(* IEC 61131-3 sources: wts-100-water-treatment-skid/plc, 4 files *)

(* ---- POU_ALARMS.st ---- *)
(*
    WTS-100  POU_ALARMS
    Alarm management.  IEC 61131-3 Structured Text.

    Implements section 6 of the control narrative, to ISA-18.2.

    FIRST OUT
    One fault usually sets off several alarms.  Supply fails, so the pump
    stops, so flow falls, so level drops, so temperature deviates.  Five
    alarms, one cause.  FIRST_OUT records whichever came first while no alarm
    was already standing, because that is the one that actually broke.
    Without it an operator at 3 a.m. faces a screen of alarms with no way to
    tell cause from consequence.

    PRIORITY
    Set by consequence and by how fast the operator must react.
    If everything is critical then nothing is.
*)

FUNCTION_BLOCK POU_ALARMS

VAR_INPUT
    ESD_01_OK       : BOOL;
    TSHH_102_OK     : BOOL;
    LSHH_102_OK     : BOOL;
    LSLL_101_OK     : BOOL;
    BOTH_PUMPS_FAIL : BOOL;
    DUTY_CHANGEOVER : BOOL;
    AIN_INVALID     : BOOL;
    AIN_STUCK       : BOOL;
    SEQ_TIMEOUT     : BOOL;
    TEMP_DEVIATION  : BOOL;
    PUMP_FB_MISMATCH: BOOL;
    DOSE_DEVIATION  : BOOL;
    ACK_CMD         : BOOL;
END_VAR

VAR_OUTPUT
    ALM_001 : BOOL;   (* emergency stop            Critical *)
    ALM_002 : BOOL;   (* over temperature          Critical *)
    ALM_003 : BOOL;   (* both raw pumps failed     Critical *)
    ALM_004 : BOOL;   (* treatment tank too full   High     *)
    ALM_005 : BOOL;   (* raw tank empty            High     *)
    ALM_006 : BOOL;   (* duty pump failed          High     *)
    ALM_007 : BOOL;   (* analog signal bad         High     *)
    ALM_008 : BOOL;   (* signal not changing       Medium   *)
    ALM_009 : BOOL;   (* sequence timeout          Medium   *)
    ALM_010 : BOOL;   (* temperature deviation     Medium   *)
    ALM_011 : BOOL;   (* pump feedback mismatch    Medium   *)
    ALM_012 : BOOL;   (* dosing deviation          Low      *)

    ANY_ALARM       : BOOL;
    ANY_UNACK       : BOOL;
    FIRST_OUT_ID    : INT;    (* 0 none, else 1..12 *)
    HIGHEST_PRIORITY: INT;    (* 0 none, 1 Critical, 2 High, 3 Medium, 4 Low *)
    ALM_HORN        : BOOL;
    ALM_BEACON      : BOOL;
END_VAR

VAR
    acked       : BOOL;
    prev_any    : BOOL;
    beacon_tick : TON;
END_VAR

(* --- alarm conditions --------------------------------------------------- *)
ALM_001 := NOT ESD_01_OK;
ALM_002 := NOT TSHH_102_OK;
ALM_003 := BOTH_PUMPS_FAIL;
ALM_004 := NOT LSHH_102_OK;
ALM_005 := NOT LSLL_101_OK;
ALM_006 := DUTY_CHANGEOVER;
ALM_007 := AIN_INVALID;
ALM_008 := AIN_STUCK;
ALM_009 := SEQ_TIMEOUT;
ALM_010 := TEMP_DEVIATION;
ALM_011 := PUMP_FB_MISMATCH;
ALM_012 := DOSE_DEVIATION;

ANY_ALARM := ALM_001 OR ALM_002 OR ALM_003 OR ALM_004 OR ALM_005 OR ALM_006
          OR ALM_007 OR ALM_008 OR ALM_009 OR ALM_010 OR ALM_011 OR ALM_012;

(* --- first out.
   --- Only captured when nothing was already standing, otherwise a later
   --- consequence would overwrite the real root cause.                  --- *)
IF ANY_ALARM AND (FIRST_OUT_ID = 0) THEN
    IF      ALM_001 THEN FIRST_OUT_ID := 1;
    ELSIF   ALM_002 THEN FIRST_OUT_ID := 2;
    ELSIF   ALM_003 THEN FIRST_OUT_ID := 3;
    ELSIF   ALM_004 THEN FIRST_OUT_ID := 4;
    ELSIF   ALM_005 THEN FIRST_OUT_ID := 5;
    ELSIF   ALM_006 THEN FIRST_OUT_ID := 6;
    ELSIF   ALM_007 THEN FIRST_OUT_ID := 7;
    ELSIF   ALM_008 THEN FIRST_OUT_ID := 8;
    ELSIF   ALM_009 THEN FIRST_OUT_ID := 9;
    ELSIF   ALM_010 THEN FIRST_OUT_ID := 10;
    ELSIF   ALM_011 THEN FIRST_OUT_ID := 11;
    ELSIF   ALM_012 THEN FIRST_OUT_ID := 12;
    END_IF;
END_IF;

IF NOT ANY_ALARM THEN
    FIRST_OUT_ID := 0;
END_IF;

(* --- highest standing priority ------------------------------------------ *)
IF   ALM_001 OR ALM_002 OR ALM_003                        THEN HIGHEST_PRIORITY := 1;
ELSIF ALM_004 OR ALM_005 OR ALM_006 OR ALM_007            THEN HIGHEST_PRIORITY := 2;
ELSIF ALM_008 OR ALM_009 OR ALM_010 OR ALM_011            THEN HIGHEST_PRIORITY := 3;
ELSIF ALM_012                                             THEN HIGHEST_PRIORITY := 4;
ELSE                                                           HIGHEST_PRIORITY := 0;
END_IF;

(* --- acknowledge.
   --- A NEW alarm clears the acknowledgement, so the horn sounds again
   --- rather than staying silent because an earlier one was acked.      --- *)
IF ANY_ALARM AND NOT prev_any THEN
    acked := FALSE;
END_IF;
prev_any := ANY_ALARM;

IF ACK_CMD THEN
    acked := TRUE;
END_IF;

IF NOT ANY_ALARM THEN
    acked := FALSE;
END_IF;

ANY_UNACK := ANY_ALARM AND NOT acked;

(* --- annunciation.
   --- Horn on any unacknowledged alarm.
   --- Beacon flashes while unacknowledged, steady once acked but still
   --- standing, so a glance tells you both things at once.              --- *)
ALM_HORN := ANY_UNACK;

beacon_tick(IN := NOT beacon_tick.Q, PT := T#500ms);
IF ANY_UNACK THEN
    ALM_BEACON := beacon_tick.Q;
ELSIF ANY_ALARM THEN
    ALM_BEACON := TRUE;
ELSE
    ALM_BEACON := FALSE;
END_IF;

END_FUNCTION_BLOCK

(* ---- POU_PUMPS.st ---- *)
(*
    WTS-100  POU_PUMPS
    Duty and standby raw water pumps.  IEC 61131-3 Structured Text.

    Same logic as the ladder drawing drawings/ladder_pumps.svg.

    Logic verified by test_ladder.py, 10 cases.
*)

FUNCTION_BLOCK POU_PUMPS

VAR_INPUT
    HS_02_START     : BOOL;   (* start pushbutton, momentary NO   *)
    HS_03_STOP_OK   : BOOL;   (* stop pushbutton, wired NC        *)
    PERM_RAW_PUMPS  : BOOL;   (* from POU_SAFETY                  *)
    XS_101A         : BOOL;   (* pump A run feedback              *)
    XS_101B         : BOOL;   (* pump B run feedback              *)
    BATCH_DONE      : BOOL;   (* one shot at end of a batch       *)
END_VAR

VAR_OUTPUT
    MTR_101A            : BOOL;
    MTR_101B            : BOOL;
    RUN_REQ             : BOOL;
    FAULT_A             : BOOL;
    FAULT_B             : BOOL;
    BOTH_PUMPS_FAILED   : BOOL;
    DUTY_IS_A           : BOOL := TRUE;
END_VAR

VAR
    tA          : TON;
    tB          : TON;
    batch_prev  : BOOL;
END_VAR

(* --- RUNG 1  start and stop with seal in.
   --- The seal in parallels the START contact ONLY.  Stop and the safety
   --- permission stay in series after it, so both can always break the rung.
   --- Putting them inside the seal in would mean the stop button does not
   --- stop the pumps once they are running.                              --- *)
RUN_REQ := (HS_02_START OR RUN_REQ) AND HS_03_STOP_OK AND PERM_RAW_PUMPS;

(* --- duty alternation.  Swap on each completed batch so running hours
   --- stay even between the two pumps.                                   --- *)
IF BATCH_DONE AND NOT batch_prev THEN
    DUTY_IS_A := NOT DUTY_IS_A;
END_IF;
batch_prev := BATCH_DONE;

(* --- RUNG 2  duty pump A                                               --- *)
MTR_101A := RUN_REQ AND DUTY_IS_A AND NOT FAULT_A;

(* --- RUNG 3  standby pump B.  Runs when B is duty, or when A has failed --- *)
MTR_101B := RUN_REQ AND NOT FAULT_B AND ((NOT DUTY_IS_A) OR FAULT_A);

(* --- RUNG 4 and 5  fault detection.
   --- Commanded on but no run feedback within 3 s means the motor did not
   --- actually start: tripped overload, failed contactor, blown fuse.    --- *)
tA(IN := MTR_101A AND NOT XS_101A, PT := T#3s);
tB(IN := MTR_101B AND NOT XS_101B, PT := T#3s);

IF tA.Q THEN FAULT_A := TRUE; END_IF;
IF tB.Q THEN FAULT_B := TRUE; END_IF;

(* --- RUNG 6  both pumps failed.  Interlock I6, trips the plant.        --- *)
BOTH_PUMPS_FAILED := FAULT_A AND FAULT_B;

END_FUNCTION_BLOCK

(* ---- POU_SAFETY.st ---- *)
(*
    WTS-100  POU_SAFETY
    Interlocks and permissives.  IEC 61131-3 Structured Text.

    This is the same logic as the ladder drawing drawings/ladder_safety.svg, written as
    text so it can be pasted straight into OpenPLC Editor and compiled.

    Runs FIRST in the scan, before the sequence and the loops, so nothing
    downstream can command an output this block has inhibited.

    All discrete safety contacts are wired normally closed.  Healthy = TRUE.
    A broken wire reads FALSE and therefore trips.

    Logic verified by test_ladder.py, 16 cases.
*)

FUNCTION_BLOCK POU_SAFETY

VAR_INPUT
    ESD_01_OK       : BOOL;   (* emergency stop not pressed      *)
    TSHH_102_OK     : BOOL;   (* below the 85 degC thermostat    *)
    XA_101A_OK      : BOOL;   (* pump A overload healthy         *)
    XA_101B_OK      : BOOL;   (* pump B overload healthy         *)
    LSLL_101_OK     : BOOL;   (* raw tank not at low low         *)
    LSHH_102_OK     : BOOL;   (* treat tank not at high high     *)
    LT_102_VALID    : BOOL;   (* level reading trustworthy       *)
    TT_102_VALID    : BOOL;   (* temperature reading trustworthy *)
    LT_102_MM       : REAL;   (* scaled treatment tank level     *)
    HS_04_RESET     : BOOL;   (* reset pushbutton                *)
END_VAR

VAR_OUTPUT
    PERM_RAW_PUMPS  : BOOL;
    PERM_HEATER     : BOOL;
    PERM_INLET      : BOOL;
    TRIP            : BOOL;
    TRIP_CAUSE      : BOOL;
    FIRST_OUT       : INT;    (* 0 none, else the interlock number *)
END_VAR

VAR
    ain_timer   : TON;
    AIN_FAULT   : BOOL;
    LVL_OK      : BOOL;
END_VAR

VAR CONSTANT
    LVL_HEATER_MIN : REAL := 800.0;
END_VAR

(* --- analog fault, interlock I7.  30 s so a brief glitch is ridden out --- *)
ain_timer(IN := NOT (LT_102_VALID AND TT_102_VALID), PT := T#30s);
AIN_FAULT := ain_timer.Q;

LVL_OK := (LT_102_MM >= LVL_HEATER_MIN);

(* --- RUNG 1  trip causes.  These are ALTERNATIVES, so OR not AND.       ---
   --- The two pump overloads are ANDed, because one failed pump changes  ---
   --- over to the standby and does not trip the plant.                   --- *)
TRIP_CAUSE :=  (NOT ESD_01_OK)
            OR (NOT TSHH_102_OK)
            OR ((NOT XA_101A_OK) AND (NOT XA_101B_OK))
            OR AIN_FAULT;

(* --- RUNG 2 and 3  latch and reset.
   --- Reset only clears the trip when the cause has already gone.        --- *)
IF TRIP_CAUSE THEN
    TRIP := TRUE;
    IF FIRST_OUT = 0 THEN
        IF    NOT ESD_01_OK                             THEN FIRST_OUT := 1;
        ELSIF NOT TSHH_102_OK                           THEN FIRST_OUT := 4;
        ELSIF (NOT XA_101A_OK) AND (NOT XA_101B_OK)     THEN FIRST_OUT := 6;
        ELSIF AIN_FAULT                                 THEN FIRST_OUT := 7;
        END_IF;
    END_IF;
ELSIF HS_04_RESET THEN
    TRIP      := FALSE;
    FIRST_OUT := 0;
END_IF;

(* --- RUNG 4  permission to run the raw water pumps.  I2 and I3.        --- *)
PERM_RAW_PUMPS := ESD_01_OK AND LSLL_101_OK AND LSHH_102_OK AND NOT TRIP;

(* --- RUNG 5  permission to run the heater.  I4 and I5.
   --- The level test uses the MEASURED level, never the sequence state,  ---
   --- so a defect in the sequence cannot fire a dry element.             --- *)
PERM_HEATER := ESD_01_OK AND TSHH_102_OK AND LT_102_VALID
               AND TT_102_VALID AND LVL_OK AND NOT TRIP;

(* --- RUNG 6  permission to open the inlet.  I3.                        --- *)
PERM_INLET := ESD_01_OK AND LSHH_102_OK AND NOT TRIP;

END_FUNCTION_BLOCK

(* ---- POU_SEQUENCE.st ---- *)
(*
    WTS-100  POU_SEQUENCE
    Batch sequence.  IEC 61131-3 Structured Text.

    IDLE -> FILL -> HEAT -> HOLD -> DISCHARGE -> DRAIN -> IDLE

    One state is active at a time.  Every transition out of every state is
    listed.  Every state has a timeout, because a state machine with no
    timeout can wait forever for a condition that will never arrive, and the
    operator gets no indication why nothing is happening.

    Any interlock forces TRIP from any state.  TRIP is latched.

    Implements section 4 of the control narrative.
*)

FUNCTION_BLOCK POU_SEQUENCE

VAR_INPUT
    START_CMD       : BOOL;
    HOLD_CMD        : BOOL;
    ABORT_CMD       : BOOL;
    AUTO_MODE       : BOOL;
    TRIP            : BOOL;     (* from POU_SAFETY *)
    PERM_INLET      : BOOL;
    PERM_HEATER     : BOOL;
    LT_101_MM       : REAL;
    LT_102_MM       : REAL;
    TT_102_C        : REAL;
    TEMP_SETPOINT   : REAL;
    RESIDENCE_S     : TIME;
END_VAR

VAR_OUTPUT
    STATE           : INT;      (* 0 IDLE 1 FILL 2 HEAT 3 HOLD
                                   4 DISCHARGE 5 DRAIN 6 TRIP 7 PAUSE *)
    RUN_PUMPS       : BOOL;
    OPEN_XV101      : BOOL;
    OPEN_XV102      : BOOL;
    ENABLE_HEATER   : BOOL;
    ENABLE_DOSING   : BOOL;
    CASCADE_ON      : BOOL;
    FLOW_SP         : REAL;
    P102_SPEED      : REAL;
    TIMEOUT_ALARM   : BOOL;
END_VAR

VAR
    t_state     : TON;
    t_stable    : TON;
    t_residence : TON;
    t_drain     : TON;
    prev_state  : INT;
    state_timeout : TIME;
    at_temp     : BOOL;
END_VAR

VAR CONSTANT
    S_IDLE      : INT := 0;
    S_FILL      : INT := 1;
    S_HEAT      : INT := 2;
    S_HOLD      : INT := 3;
    S_DISCHARGE : INT := 4;
    S_DRAIN     : INT := 5;
    S_TRIP      : INT := 6;
    S_PAUSE     : INT := 7;
END_VAR

(* --- a trip beats everything, from any state --------------------------- *)
IF TRIP THEN
    STATE := S_TRIP;
END_IF;

(* --- pick the timeout for the state we are in.
   --- Rule: two to three times the expected duration.  Too tight and it
   --- nuisance trips on a slow day, too loose and a real fault goes
   --- unnoticed far too long.                                           --- *)
CASE STATE OF
    S_FILL:      state_timeout := T#900s;    (* fill takes about 5 min   *)
    S_HEAT:      state_timeout := T#5400s;   (* heat takes about 45 min  *)
    S_DISCHARGE: state_timeout := T#600s;
ELSE
    state_timeout := T#0s;
END_CASE;

t_state(IN := (STATE <> prev_state), PT := T#1s);
IF STATE <> prev_state THEN
    t_state(IN := FALSE);
END_IF;
prev_state := STATE;

CASE STATE OF

(* ------------------------------------------------------------ 4.0 IDLE *)
S_IDLE:
    RUN_PUMPS     := FALSE;
    OPEN_XV101    := FALSE;
    OPEN_XV102    := FALSE;
    ENABLE_HEATER := FALSE;
    ENABLE_DOSING := FALSE;
    CASCADE_ON    := FALSE;
    FLOW_SP       := 0.0;
    P102_SPEED    := 0.0;

    (* the raw tank check stops a batch that is guaranteed to fail *)
    IF START_CMD AND AUTO_MODE AND NOT TRIP AND (LT_101_MM > 400.0) THEN
        STATE := S_FILL;
    END_IF;

(* ------------------------------------------------------------ 4.1 FILL *)
S_FILL:
    OPEN_XV101 := PERM_INLET;
    RUN_PUMPS  := TRUE;
    CASCADE_ON := FALSE;      (* fixed flow: no level worth controlling yet *)
    FLOW_SP    := 30.0;

    IF LT_102_MM >= 1200.0 THEN
        STATE := S_HEAT;
    END_IF;

(* ------------------------------------------------------------ 4.2 HEAT *)
S_HEAT:
    OPEN_XV101    := PERM_INLET;
    RUN_PUMPS     := TRUE;
    CASCADE_ON    := TRUE;    (* level loop now sets the flow setpoint *)
    ENABLE_HEATER := PERM_HEATER;
    ENABLE_DOSING := TRUE;

    (* must sit within band CONTINUOUSLY, so a momentary excursion through
       setpoint while the tank is still stratified does not advance us *)
    at_temp := ABS(TT_102_C - TEMP_SETPOINT) <= 0.5;
    t_stable(IN := at_temp, PT := T#60s);

    IF t_stable.Q THEN
        STATE := S_HOLD;
    END_IF;

(* ------------------------------------------------------------ 4.3 HOLD *)
S_HOLD:
    CASCADE_ON    := TRUE;
    ENABLE_HEATER := PERM_HEATER;
    ENABLE_DOSING := TRUE;

    t_residence(IN := TRUE, PT := RESIDENCE_S);
    IF t_residence.Q THEN
        STATE := S_DISCHARGE;
    END_IF;

(* ------------------------------------------------------- 4.4 DISCHARGE *)
S_DISCHARGE:
    ENABLE_HEATER := FALSE;   (* heater OFF before the tank starts emptying *)
    ENABLE_DOSING := FALSE;
    RUN_PUMPS     := FALSE;
    OPEN_XV101    := FALSE;
    CASCADE_ON    := FALSE;
    OPEN_XV102    := TRUE;
    P102_SPEED    := 60.0;

    IF LT_102_MM <= 300.0 THEN
        STATE := S_DRAIN;
    END_IF;

(* ----------------------------------------------------------- 4.5 DRAIN *)
S_DRAIN:
    OPEN_XV102 := TRUE;
    P102_SPEED := 100.0;

    (* 10 s confirmation, so a splash as the last liquid clears the tapping
       does not end the batch early *)
    t_drain(IN := (LT_102_MM <= 50.0), PT := T#10s);
    IF t_drain.Q THEN
        OPEN_XV102 := FALSE;
        P102_SPEED := 0.0;
        STATE      := S_IDLE;
    END_IF;

(* ------------------------------------------------------------ 4.7 TRIP *)
S_TRIP:
    RUN_PUMPS     := FALSE;
    OPEN_XV101    := FALSE;
    OPEN_XV102    := FALSE;
    ENABLE_HEATER := FALSE;
    ENABLE_DOSING := FALSE;
    CASCADE_ON    := FALSE;
    FLOW_SP       := 0.0;
    P102_SPEED    := 0.0;

    IF NOT TRIP THEN
        STATE := S_IDLE;
    END_IF;

(* ----------------------------------------------------------- 4.6 PAUSE *)
S_PAUSE:
    RUN_PUMPS     := FALSE;
    ENABLE_HEATER := FALSE;
    FLOW_SP       := 0.0;
    IF START_CMD THEN
        STATE := S_HOLD;
    END_IF;

END_CASE;

(* --- operator hold, from any running state ----------------------------- *)
IF HOLD_CMD AND (STATE > S_IDLE) AND (STATE < S_TRIP) THEN
    STATE := S_PAUSE;
END_IF;

(* --- 4.8 controlled stop.  Order matters: heater first, valves last,
   --- so the heater is never energised in a tank being emptied.        --- *)
IF ABORT_CMD THEN
    ENABLE_HEATER := FALSE;
    ENABLE_DOSING := FALSE;
    RUN_PUMPS     := FALSE;
    OPEN_XV101    := FALSE;
    OPEN_XV102    := FALSE;
    STATE         := S_IDLE;
END_IF;

(* --- state timeout ------------------------------------------------------ *)
TIMEOUT_ALARM := (state_timeout > T#0s) AND t_state.ET > state_timeout;
IF TIMEOUT_ALARM THEN
    STATE := S_DRAIN;
END_IF;

END_FUNCTION_BLOCK
